# EPICS autosave request: iocBoot/iocTomoScan_6BM/auto_settings.req
file "tomoScan_settings.req", P=$(P), R=$(R)
file "tomoScan_PSO_settings.req", P=$(P), R=$(R)
file "tomoScan_6BM_settings.req", P=$(P), R=$(R)
